// TIA Portal V20 export
TYPE "TrackingData"
// stored: Namespace LineD1
   STRUCT
      Barcode : String;
      ResponseCode : UInt;
      HeightLimit : Bool;
      ActualWeight : Struct
         inRealValue : Real;
         inStringFormat : String;
      END_STRUCT;
      EXIT_1_ : Array[1..1] of Bool;
      EXIT_2_ : Array[1..6] of Bool;
      ToteDir : "LineD1.ItemDir";
   END_STRUCT;
END_TYPE
